FUNCTION_BLOCK WoodBunkEx EXTENDS SectionEx
VAR_IN_OUT
	A21_LSC_C21 : ConveyorLSC;
END_VAR
VAR_IN_OUT
	robotLeft, robotRight : RobotA21;
	toolStorageLeft, toolStorageRight : A21ToolStorage;
	
	stagingTableLeft, stagingTableRight : StagingTable;
	magazineLeft, magazineRight : SkidMagazine;
	
	strapper : StrapMachine;
	
	insertionLeft, insertionRight : Insertion;
	pistonBottom : SimplePiston;
	
	suctionTop : ARRAY[*] OF SuctionPad; (*1..3*)
	suctionLeft : ARRAY[*] OF SuctionPad; (*1..4*)
	suctionRight : ARRAY[*] OF SuctionPad; (*1..4*)
	suctionBottom : ARRAY[*] OF SuctionPad; (*1..2*)
END_VAR
VAR
	conveyorPos : REAL; //may need to move this to SectionEx
	
	step : (IDLE, STAGING, LOAD_WB, PUSH, STRAP, RELEASE, COMPLETE := 1050);
	
	stageStepLeft, stageStepRight : INT;
	loadStepLeft, loadStepRight : INT;
END_VAR
VAR //bundle data
	demoHeight : REAL := 640; //mm
	materialsArr : (*REFERENCE TO*) ARRAY[0..Consts.maxPairs] OF PositionMaterials;
END_VAR
VAR
	//AOIs encapsulate functionality and reduce the number of module variables
	aoiTemplateLeft, aoiTemplateRight : AOI_StagingTemplate;
	aoiStageLeft, aoiStageRight : AOI_StageWoodBunk; 
	aoiLoadLeft, aoiLoadRight : AOI_LoadWoodBunk;
	
	suctionRelease : TON;
	
	//for testing, to be removed when deployoed
	latchLeft, latchRight : BOOL; //prevents SMC sliders from overshooting
	suctionEnableTop, suctionEnableLeft, suctionEnableRight, suctionEnableBottom : BOOL;
END_VAR

aoiBlocks();

SUPER^();

(*
any PackML state-methods that SectionEx has a concrete implementation for will be overriden by concrete FBs that extend it
(ie: all or most of them)

to call the base implementation, add:
	SUPER^.ps_<state>();
to the concrete FB's implementation of that state-method
*)

METHOD PROTECTED aoiBlocks : BOOL
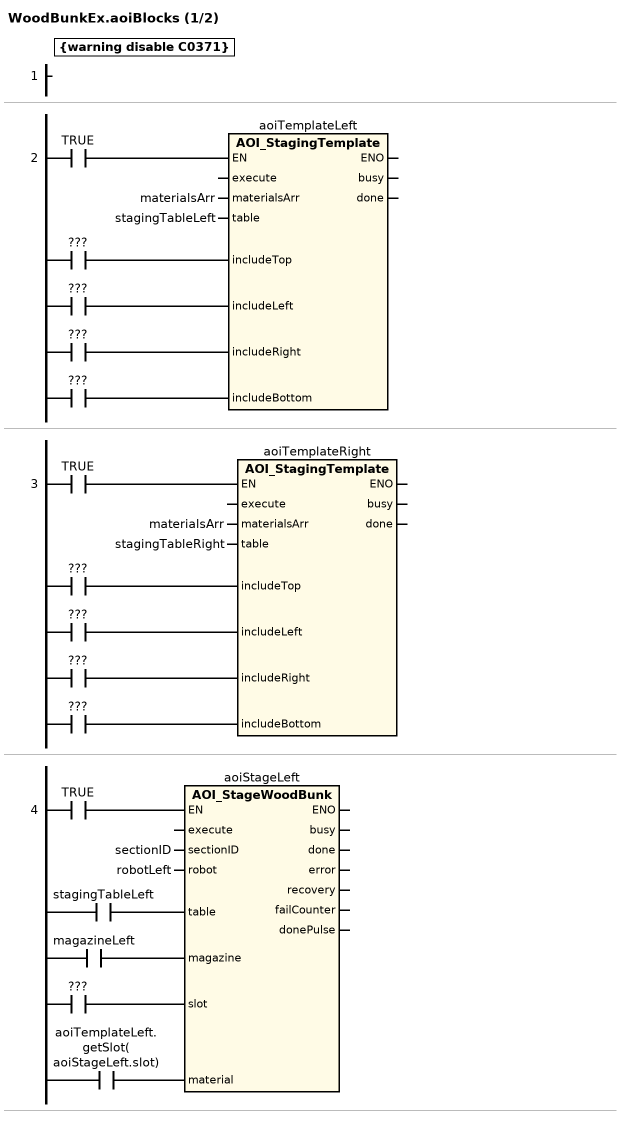
// NETWORK 1
// label: {warning disable C0371}

// NETWORK 2
aoiTemplateLeft(materialsArr := materialsArr, table := stagingTableLeft); // AOI_StagingTemplate

// NETWORK 3
aoiTemplateRight(materialsArr := materialsArr, table := stagingTableRight); // AOI_StagingTemplate

// NETWORK 4
aoiStageLeft(
    sectionID := sectionID,
    robot := robotLeft,
    table := stagingTableLeft,
    magazine := magazineLeft,
    material := aoiTemplateLeft.getSlot(aoiStageLeft.slot)); // AOI_StageWoodBunk

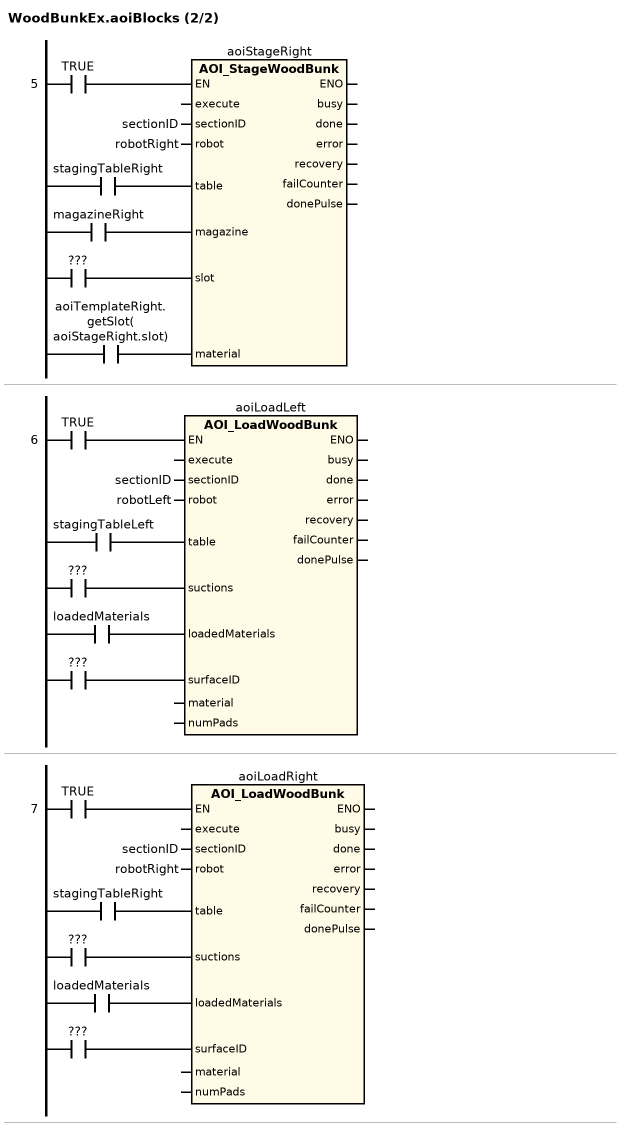
// NETWORK 5
aoiStageRight(
    sectionID := sectionID,
    robot := robotRight,
    table := stagingTableRight,
    magazine := magazineRight,
    material := aoiTemplateRight.getSlot(aoiStageRight.slot)); // AOI_StageWoodBunk

// NETWORK 6
aoiLoadLeft(
    sectionID := sectionID,
    robot := robotLeft,
    table := stagingTableLeft,
    loadedMaterials := loadedMaterials); // AOI_LoadWoodBunk

// NETWORK 7
aoiLoadRight(
    sectionID := sectionID,
    robot := robotRight,
    table := stagingTableRight,
    loadedMaterials := loadedMaterials); // AOI_LoadWoodBunk
END_METHOD

METHOD PROTECTED load : BOOL
VAR_INPUT
	pairIndex : INT;
END_VAR
VAR_OUTPUT
	error : BOOL;
END_VAR
VAR
	pair : REFERENCE TO PositionMaterials REF= materialsArr[pairIndex];
	errorLeft, errorRight : BOOL;
END_VAR
{warning disable C0371}
(*
this is the new code for loading wood bunks from staging table to insertion
loading sequences are independent as each side has its own step variable
can be extended by changing the include<> parameters
*)

load :=
	loadEx(
		robot:= robotLeft, 
		aoiLoad:= aoiLoadLeft, 
		loadStep:= loadStepLeft, 
		pairIndex:= pairIndex, 
		includeTop:= TRUE, 
		includeLeft:= TRUE, 
		includeRight:= FALSE, 
		includeBottom:= FALSE, 
		error=> errorLeft)
	AND
	loadEx(
		robot:= robotRight, 
		aoiLoad:= aoiLoadRight, 
		loadStep:= loadStepRight, 
		pairIndex:= pairIndex, 
		includeTop:= FALSE, 
		includeLeft:= FALSE, 
		includeRight:= TRUE, 
		includeBottom:= TRUE, 
		error=> errorRight);
		
error := errorLeft OR errorRight;

(*
below is the old code for loading wood bunks from staging table to insertion
it loads wood bunks in sets - top/bottom, then sides
if one side is finished loading a set before the other, it waits until the other side is done before advancing the set
*)
(*
IF robotLeft.error OR robotRight.error THEN
	error := TRUE;
	RETURN;
	
ELSIF 
	(robotLeft.reservation <> sectionID AND_THEN NOT robotLeft.reserve(sectionID)) OR 
	(robotRight.reservation <> sectionID AND_THEN NOT robotRight.reserve(sectionID))
THEN //loading requires both robots be reserved together
	RETURN;
	
ELSIF //robots have wrong tool
	(robotLeft.tool <> sectionID AND_THEN NOT robotLeft.changeEOAT(targetTool := sectionID)) OR
	(robotRight.tool <> sectionID AND_THEN NOT robotRight.changeEOAT(targetTool := sectionID))
THEN
	RETURN;
	
END_IF

CASE loadStep OF
	0: //top and bottom
		IF aoiLoadLeft.done AND aoiLoadRight.done THEN
			aoiLoadLeft.execute := aoiLoadRight.execute := FALSE;
			aoiLoadLeft.material := aoiLoadRight.material := '';
			
			aoiLoadLeft.reset();
			aoiLoadRight.reset();
			loadStep := 10;
			RETURN;
		END_IF
		
		aoiLoadLeft.suctions := suctionTop;
		aoiLoadLeft.surfaceID := Surface.TOP;
		aoiLoadLeft.material := pair.top;
		aoiLoadLeft.numPads := UPPER_BOUND(suctionTop, 1) - LOWER_BOUND(suctionTop, 1) + 1;
		
		aoiLoadRight.suctions := suctionBottom;
		aoiLoadRight.surfaceID := Surface.BOTTOM;
		aoiLoadRight.material := pair.bottom;
		aoiLoadRight.numPads := UPPER_BOUND(suctionBottom, 1) - LOWER_BOUND(suctionBottom, 1) + 1;
		
		aoiLoadLeft.execute := NOT aoiLoadLeft.done AND NOT aoiLoadLeft.busy;
		aoiLoadRight.execute := NOT aoiLoadRight.done AND NOT aoiLoadRight.busy;
		
	10: //sides
		IF aoiLoadLeft.done AND aoiLoadRight.done THEN
			aoiLoadLeft.execute := aoiLoadRight.execute := FALSE;
			aoiLoadLeft.material := aoiLoadRight.material := '';
			
			aoiLoadLeft.reset();
			aoiLoadRight.reset();
			loadStep := COMPLETE;
			RETURN;
		END_IF
		
		aoiLoadLeft.suctions := suctionLeft;
		aoiLoadLeft.surfaceID := Surface.LEFT;
		aoiLoadLeft.material := pair.left;
		aoiLoadLeft.numPads := UPPER_BOUND(suctionLeft, 1) - LOWER_BOUND(suctionLeft, 1) + 1;
		
		aoiLoadRight.suctions := suctionRight;
		aoiLoadRight.surfaceID := Surface.RIGHT;
		aoiLoadRight.material := pair.right;
		aoiLoadRight.numPads := UPPER_BOUND(suctionRight, 1) - LOWER_BOUND(suctionRight, 1) + 1;
		
		aoiLoadLeft.execute := NOT aoiLoadLeft.done AND NOT aoiLoadLeft.busy;
		aoiLoadRight.execute := NOT aoiLoadRight.done AND NOT aoiLoadRight.busy;
		
	COMPLETE:				
		robotLeft.release(sectionID);
		robotRight.release(sectionID);
		
		aoiLoadLeft.material := aoiLoadRight.material := '';
		aoiLoadLeft.execute := aoiLoadRight.execute := FALSE;
		
		loadStep := 0;
		load := TRUE;
END_CASE

//--------------------------------------------------
IF aoiLoadLeft.recovery THEN //if loading in recovery mode - refill table, resume loading when finished
	aoiLoadLeft.execute := stageEx(
		robot:= robotLeft, 
		aoiTemplate:= aoiTemplateLeft, 
		aoiStaging:= aoiStageLeft, 
		stageStep:= stageStepLeft, 
		includeTop:= TRUE, 
		includeLeft:= TRUE, 
		includeRight:= FALSE, 
		includeBottom:= FALSE, 
		error=> );
ELSE
	//loadLeft.execute := NOT loadLeft.busy AND NOT loadLeft.done;
END_IF
//--------------------------------------------------
IF aoiLoadRight.recovery THEN
	aoiLoadRight.execute := stageEx(
		robot:= robotRight, 
		aoiTemplate:= aoiTemplateRight, 
		aoiStaging:= aoiStageRight, 
		stageStep:= stageStepRight, 
		includeTop:= FALSE, 
		includeLeft:= FALSE, 
		includeRight:= TRUE, 
		includeBottom:= TRUE, 
		error=> );
ELSE
	//loadRight.execute := NOT loadRight.busy AND NOT loadRight.done;
END_IF
//--------------------------------------------------
	
error := aoiLoadLeft.error OR aoiLoadRight.error;
*)
END_METHOD

METHOD PRIVATE loadEx : BOOL
VAR_IN_OUT
	robot : RobotA21;
	aoiLoad : AOI_LoadWoodBunk;
	loadStep : INT;
END_VAR
VAR_INPUT
	pairIndex : INT;
	includeTop, includeLeft, includeRight, includeBottom : BOOL;
END_VAR
VAR_OUTPUT
	error : BOOL;
END_VAR
VAR
	pair : REFERENCE TO PositionMaterials REF= materialsArr[pairIndex];
END_VAR
{warning disable C0371}
IF robot.error THEN
	error := TRUE;
	RETURN;
ELSIF robot.reservation <> sectionID AND_THEN NOT robot.reserve(sectionID) THEN
	RETURN;
ELSIF robot.tool <> sectionID AND_THEN NOT robot.changeEOAT(targetTool := sectionID) THEN
	RETURN;
END_IF

error := aoiLoad.error;

CASE loadStep OF
	0:
		loadStep := Surface.TOP;
	
	Surface.TOP:		
		IF NOT includeTop OR aoiLoad.donePulse THEN
			aoiLoad.execute := FALSE;
			aoiLoad.material := '';
			loadStep := Surface.BOTTOM;
			RETURN;
		END_IF
		
		aoiLoad.surfaceID := Surface.TOP;
		aoiLoad.material := pair.top;
		aoiLoad.suctions := suctionTop;
		aoiLoad.numPads := UPPER_BOUND(suctionTop, 1) - LOWER_BOUND(suctionTop, 1) + 1;
		
		aoiLoad.execute := NOT aoiLoad.busy;
		
	Surface.BOTTOM:
		IF NOT includeBottom OR aoiLoad.donePulse THEN
			aoiLoad.execute := FALSE;
			aoiLoad.material := '';
			loadStep := Surface.LEFT;
			RETURN;
		END_IF
		
		aoiLoad.surfaceID := Surface.BOTTOM;
		aoiLoad.material := pair.bottom;
		aoiLoad.suctions := suctionBottom;
		aoiLoad.numPads := UPPER_BOUND(suctionBottom, 1) - LOWER_BOUND(suctionBottom, 1) + 1;
		
		aoiLoad.execute := NOT aoiLoad.busy;
		
	Surface.LEFT:
		IF NOT includeLeft OR aoiLoad.donePulse THEN
			aoiLoad.execute := FALSE;
			aoiLoad.material := '';
			loadStep := Surface.RIGHT;
			RETURN;
		END_IF
		
		aoiLoad.surfaceID := Surface.LEFT;
		aoiLoad.material := pair.left;
		aoiLoad.suctions := suctionLeft;
		aoiLoad.numPads := UPPER_BOUND(suctionLeft, 1) - LOWER_BOUND(suctionLeft, 1) + 1;
		
		aoiLoad.execute := NOT aoiLoad.busy;
		
	Surface.RIGHT:
		IF NOT includeRight OR aoiLoad.donePulse THEN
			aoiLoad.execute := FALSE;
			aoiLoad.material := '';
			loadStep := COMPLETE;
			RETURN;
		END_IF
		
		aoiLoad.surfaceID := Surface.RIGHT;
		aoiLoad.material := pair.right;
		aoiLoad.suctions := suctionRight;
		aoiLoad.numPads := UPPER_BOUND(suctionRight, 1) - LOWER_BOUND(suctionRight, 1) + 1;
		
		aoiLoad.execute := NOT aoiLoad.busy;
		
	COMPLETE:				
		robot.release(sectionID);
		
		aoiLoad.material := '';
		aoiLoad.execute := FALSE;
		
		loadEx := TRUE;
END_CASE
END_METHOD

METHOD PROTECTED maintenance : BOOL
VAR_INPUT
END_VAR
{warning disable C0371}
//no specific tasks yet, free run and testing
SetSuctions(suctionTop, suctionEnableTop);
SetSuctions(suctionLeft, suctionEnableLeft);
SetSuctions(suctionRight, suctionEnableRight);
SetSuctions(suctionBottom, suctionEnableBottom);

IF robotLeft.Done THEN
	robotLeft.clearCommand();
END_IF

IF robotRight.Done THEN
	robotRight.clearCommand();
END_IF
END_METHOD

METHOD PROTECTED manual : BOOL
VAR_INPUT
END_VAR
END_METHOD

METHOD PROTECTED process : BOOL
VAR_INPUT
	auto : BOOL;
END_VAR
VAR_OUTPUT
	error : BOOL;
END_VAR
VAR
	currentPair : REFERENCE TO PositionMaterials REF= materialsArr[iPair];
END_VAR
{warning disable C0371}
IF iPair >= Consts.maxPairs THEN
	process := TRUE;
	RETURN;
ELSIF NOT PositionIsValid(pair := currentPair) THEN
	iPair := iPair + 1;
	RETURN;
END_IF

CASE step OF
	IDLE:
		IF auto OR_ELSE execute THEN
			step := STAGING;
		END_IF

	LOAD_WB:
		IF
			directionCheckAndSet(conveyorPos, currentPair.position) AND 
			( (auto AND done) OR_ELSE (NOT auto AND execute) )
		THEN
			robotLeft.clearCommand();
			robotRight.clearCommand();
			
			aoiLoadLeft.reset();
			aoiLoadRight.reset();
			
			loadStepLeft := loadStepRight := 0;
			stageStepLeft := stageStepRight := 0;
			
			done := FALSE;
			suctionEnableTop := suctionEnableLeft := suctionEnableRight := suctionEnableBottom := FALSE;
			execute := FALSE;
			
			step := PUSH;
			RETURN;
		END_IF
		
		IF NOT done THEN
			done := load(pairIndex := iPair, error => error);
		END_IF
		
		IF NOT auto THEN
			SetSuctions(suctionTop, suctionEnableTop);
			SetSuctions(suctionLeft, suctionEnableLeft);
			SetSuctions(suctionRight, suctionEnableRight);
			SetSuctions(suctionBottom, suctionEnableBottom);
		END_IF
		
	PUSH:
		IF
			(auto AND latchLeft AND latchRight AND pistonBottom.extended) OR_ELSE
			(NOT auto AND execute)
		THEN
			insertionLeft.stop();
			insertionRight.stop();
			
			latchLeft := latchRight := FALSE;
			execute := FALSE;
			step := STRAP;
			RETURN;
		END_IF
		
		IF NOT validateInsertion(checkTop:= FALSE, checkLeft:= FALSE, checkRight:= FALSE, checkBottom:= FALSE) THEN
			error := TRUE;
			RETURN;
		END_IF
		
		IF 
			insertionLeft.sliderPos <> demoHeight/2 OR 
			insertionRight.sliderPos <> demoHeight/2
		THEN
			insertionLeft.align(demoHeight/2);
			insertionRight.align(demoHeight/2);
			RETURN;
		END_IF
		
		
		IF insertionLeft.Contact THEN
			latchLeft := TRUE;
		ELSIF NOT latchLeft THEN
			insertionLeft.press();
		END_IF
		
		IF insertionRight.Contact THEN
			latchRight := TRUE;
		ELSIF NOT latchRight THEN
			insertionRight.press();
		END_IF
		pistonBottom.extend();
		
	STRAP:
		suctionRelease(IN:= , PT:= suctionReleaseDelay, Q=> , ET=> );
		
		strapper.bEnable := TRUE;
		IF strapper.done THEN
			suctionRelease.IN := FALSE;
			step := RELEASE;
			RETURN;
		END_IF
		
		IF suctionRelease.Q THEN
			SetSuctions(suctionTop, FALSE);
			SetSuctions(suctionLeft, FALSE);
			SetSuctions(suctionRight, FALSE);
			SetSuctions(suctionBottom, FALSE);
		ELSIF strapper.atBundleLevel THEN
			suctionRelease.IN := TRUE;
		END_IF
		
		IF strapper.ready THEN
			strapper.strap();
		END_IF
		
		IF execute THEN
			suctionRelease.IN := FALSE;
			execute := FALSE;
			step := RELEASE;
		END_IF
		
	RELEASE: //release command		
		insertionLeft.toHome();
		insertionRight.toHome();
		pistonBottom.retract();
		
		IF 
			(insertionLeft.screw.AtHome AND insertionRight.screw.AtHome AND pistonBottom.retracted) OR
			execute
		THEN
			execute := FALSE;
			step := COMPLETE;
		END_IF
	
	COMPLETE:
		//reset everything
		iPair := iPair + 1;
		step := IDLE;
END_CASE
END_METHOD

METHOD PROTECTED ps_AbortCondition : BOOL
VAR_INPUT
END_VAR
{warning disable C0371}
ps_AbortCondition :=
	insertionLeft.error OR 
	insertionRight.error OR 
	robotLeft.error OR 
	robotRight.error OR
	strapper.error;
END_METHOD

METHOD PROTECTED ps_Aborted : BOOL
VAR_INPUT
END_VAR
ps_Aborted := TRUE;
END_METHOD

METHOD PROTECTED ps_Aborting : BOOL
VAR_INPUT
END_VAR
{warning disable C0371}
insertionLeft.stop();
insertionRight.stop();
pistonBottom.stop();

aoiLoadLeft.reset();
aoiLoadRight.reset();

aoiStageLeft.reset();
aoiStageRight.reset();

robotLeft.clearCommand();
robotRight.clearCommand();

//stop conveyors

ps_Aborting :=
	NOT insertionLeft.active AND
	NOT insertionRight.active AND
	NOT pistonBottom.busy AND
	NOT robotLeft.Busy AND
	NOT robotRight.Busy;
END_METHOD

METHOD PROTECTED ps_Clearing : BOOL
VAR_INPUT
END_VAR
{warning disable C0371}
insertionLeft.reset();
insertionRight.reset();

ps_Clearing := 
	NOT insertionLeft.error AND
	NOT insertionRight.error AND
	NOT strapper.error AND
	NOT robotLeft.error AND
	NOT robotRight.error;
END_METHOD

METHOD PROTECTED ps_Complete : BOOL
VAR_INPUT
END_VAR
ps_Complete := TRUE;
END_METHOD

METHOD PROTECTED ps_Completing : BOOL
VAR_INPUT
END_VAR
ps_Completing := NOT occupied;
END_METHOD

METHOD PROTECTED ps_Execute : BOOL
VAR_INPUT
END_VAR
VAR_OUTPUT
	error : BOOL;
END_VAR
SUPER^.ps_Execute();
END_METHOD

METHOD PROTECTED ps_Held : BOOL
VAR_INPUT
END_VAR
ps_Held := NOT hold;
END_METHOD

METHOD PROTECTED ps_HoldCondition : BOOL
VAR_INPUT
END_VAR
END_METHOD

METHOD PROTECTED ps_Holding : BOOL
VAR_INPUT
END_VAR
{warning disable C0371}
insertionLeft.stop();
insertionRight.stop();
pistonBottom.stop();
//set robot to pause

ps_Holding :=
	NOT insertionLeft.active AND
	NOT insertionRight.active;
END_METHOD

METHOD PROTECTED ps_Idle : BOOL
VAR_INPUT
END_VAR
ps_Idle := execute;
execute := FALSE;
END_METHOD

METHOD PROTECTED ps_Resetting : BOOL
VAR_INPUT
END_VAR
{warning disable C0371}
insertionLeft.reset();
insertionRight.reset();

ps_Resetting := 
	reset AND
	NOT insertionLeft.error AND
	NOT insertionRight.error AND
	NOT strapper.error AND
	NOT robotLeft.error AND
	NOT robotRight.error;
END_METHOD

METHOD PROTECTED ps_Starting : BOOL
VAR_INPUT
END_VAR
{warning disable C0371}
robotLeft.clearCommand();
robotRight.clearCommand();

insertionLeft.homingSequence();
insertionRight.homingSequence();
pistonBottom.retract();

ps_Starting := 
	insertionLeft.screw.HomeSet AND 
	insertionRight.screw.HomeSet AND 
	pistonBottom.retracted;
END_METHOD

METHOD PROTECTED ps_StopCondition : BOOL
VAR_INPUT
END_VAR
ps_StopCondition := 
	stop;
END_METHOD

METHOD PROTECTED ps_Stopped : BOOL
VAR_INPUT
END_VAR
ps_Stopped := TRUE;
END_METHOD

METHOD PROTECTED ps_Stopping : BOOL
VAR_INPUT
END_VAR
{warning disable C0371}
insertionLeft.stop();
insertionRight.stop();
pistonBottom.stop();

aoiLoadLeft.reset();
aoiLoadRight.reset();

aoiStageLeft.reset();
aoiStageRight.reset();

robotLeft.clearCommand();
robotRight.clearCommand();

//stop conveyors

ps_Stopping :=
	NOT insertionLeft.active AND
	NOT insertionRight.active AND
	NOT pistonBottom.busy AND
	NOT robotLeft.Busy AND
	NOT robotRight.Busy;
END_METHOD

METHOD PROTECTED ps_SuspendCondition : BOOL
VAR_INPUT
END_VAR
END_METHOD

METHOD PROTECTED ps_Suspended : BOOL
VAR_INPUT
END_VAR
ps_Suspended := NOT ps_SuspendCondition();
END_METHOD

METHOD PROTECTED ps_Suspending : BOOL
VAR_INPUT
END_VAR
ps_Suspending := TRUE;
END_METHOD

METHOD PROTECTED ps_Unholding : BOOL
VAR_INPUT
END_VAR
ps_Unholding := TRUE;
END_METHOD

METHOD PROTECTED ps_Unsuspending : BOOL
VAR_INPUT
END_VAR
ps_Unsuspending := TRUE;
END_METHOD

METHOD PROTECTED FINAL runSectionTasks : BOOL
VAR_INPUT
	auto : BOOL;
END_VAR
VAR_OUTPUT
	error : BOOL;
END_VAR
SUPER^.runSectionTasks(auto := auto, error => error);

CASE status OF //add additional instructions for each state
	SectionTask.IDLE:
		//
	
	SectionTask.ALIGNING:
		stage(error => error);
		
	SectionTask.ACTIVE:
		//
		
	SectionTask.CLEARING:
		aoiLoadLeft.reset();
		aoiLoadRight.reset();
		
		aoiStageLeft.reset();
		aoiStageRight.reset();
		
		aoiTemplateLeft.reset();
		aoiTemplateRight.reset();
		
	SectionTask.COMPLETE:	
		//
		
	-100:
		//
		
END_CASE
END_METHOD

METHOD PROTECTED stage : BOOL
VAR_OUTPUT
	error : BOOL;
END_VAR
{warning disable C0371}

(*
this method only exists to call stageEx() for both robots
*)
(*
stage := leftDone AND rightDone;

IF NOT leftDone THEN
	leftDone := stageEx(
		robot:= robotLeft, 
		aoiTemplate:= aoiTemplateLeft, 
		aoiStaging:= aoiStageLeft, 
		stageStep:= stageStepLeft, 
		//iSlot:= iSlotLeft, 
		includeTop:= TRUE, 
		includeLeft:= TRUE, 
		includeRight:= FALSE, 
		includeBottom:= FALSE, 
		error=> );
END_IF

IF NOT rightDone THEN
	rightDone := stageEx(
		robot:= robotRight, 
		aoiTemplate:= aoiTemplateRight, 
		aoiStaging:= aoiStageRight, 
		stageStep:= stageStepRight, 
		//iSlot:= iSlotRight, 
		includeTop:= FALSE, 
		includeLeft:= FALSE, 
		includeRight:= TRUE, 
		includeBottom:= TRUE, 
		error=> );
END_IF
*)

stage := 
	stageEx(
		robot:= robotLeft, 
		aoiTemplate:= aoiTemplateLeft, 
		aoiStaging:= aoiStageLeft, 
		stageStep:= stageStepLeft, 
		includeTop:= TRUE, 
		includeLeft:= TRUE, 
		includeRight:= FALSE, 
		includeBottom:= FALSE, 
		error=> )
	AND
	stageEx(
		robot:= robotRight, 
		aoiTemplate:= aoiTemplateRight, 
		aoiStaging:= aoiStageRight, 
		stageStep:= stageStepRight, 
		includeTop:= FALSE, 
		includeLeft:= FALSE, 
		includeRight:= TRUE, 
		includeBottom:= TRUE, 
		error=> );
END_METHOD

METHOD PRIVATE stageEx : BOOL
VAR_IN_OUT
	robot : RobotA21;
	aoiTemplate : AOI_StagingTemplate;
	aoiStaging : AOI_StageWoodBunk;
	stageStep : INT;
END_VAR
VAR_INPUT
	includeTop, includeLeft, includeRight, includeBottom : BOOL;
END_VAR
VAR_OUTPUT
	error : BOOL;
END_VAR
{warning disable C0371}
IF robot.error THEN
	error := TRUE;
	RETURN;
ELSIF robot.reservation <> sectionID AND_THEN NOT robot.reserve(sectionID) THEN
	RETURN;
ELSIF robot.tool <> sectionID AND_THEN NOT robot.changeEOAT(targetTool := sectionID) THEN
	RETURN;
END_IF

CASE stageStep OF
	0: //generate staging template
		IF aoiTemplate.done THEN
			aoiTemplate.execute := FALSE;
			stageStep := 10;
			RETURN;
		END_IF
		
		aoiTemplate.execute := NOT aoiTemplate.busy;
		
		aoiTemplate.includeTop := includeTop;
		aoiTemplate.includeLeft := includeLeft;
		aoiTemplate.includeRight := includeRight;
		aoiTemplate.includeBottom := includeBottom;
		
	10: //stage tables
		IF aoiStaging.slot > 10 THEN
			aoiStaging.execute := FALSE;			
			stageStep := COMPLETE;
			RETURN;
		END_IF
		
		aoiStaging.execute := NOT aoiStaging.busy; //execute if aoiStaging is ready
		
		aoiStaging.slot := MAX(1, aoiStaging.slot); //if 0, sets to 1
		aoiStaging.slot := MIN(aoiStaging.slot, 999); //prevents overflow 
		
		IF aoiStaging.donePulse THEN
			aoiStaging.slot := aoiStaging.slot + 1;
		END_IF
	
	COMPLETE:
		aoiTemplate.clearTemplate();
		aoiTemplate.execute := FALSE;
		aoiStaging.execute := FALSE;
		aoiStaging.reset();
		
		robot.release(sectionID);
		
		aoiStaging.slot := 0;
		
		stageEx := TRUE;
		//stageStep := 0;
END_CASE

error := aoiStaging.error;
END_METHOD

METHOD PROTECTED unload : BOOL
VAR_INPUT
END_VAR
//unload from insertion
//remove from staging table
END_METHOD

METHOD PROTECTED validateInsertion : BOOL
VAR_INPUT
	checkTop : BOOL;
	checkLeft : BOOL;
	checkRight : BOOL;
	checkBottom : BOOL;
END_VAR
validateInsertion := 
	(NOT checkTop OR_ELSE SuctionQuality(suctions:= suctionTop)) AND
	(NOT checkLeft OR_ELSE SuctionQuality(suctions:= suctionLeft)) AND
	(NOT checkRight OR_ELSE SuctionQuality(suctions:= suctionRight)) AND
	(NOT checkBottom OR_ELSE SuctionQuality(suctions:= suctionBottom));

(*
validateSuctionQuality := 
	(
		NOT checkTop OR_ELSE InsertionQuality(
			suctions:= suctionTop, 
			insertionMaterial:= loadedMaterials[Surface.TOP], 
			recipeMaterial:= materialsArr[iPair].top)
	) AND
	(
		NOT checkLeft OR_ELSE InsertionQuality(
			suctions:= suctionLeft, 
			insertionMaterial:= loadedMaterials[Surface.LEFT], 
			recipeMaterial:= materialsArr[iPair].left)
	) AND
	(
		NOT checkRight OR_ELSE InsertionQuality(
			suctions:= suctionRight, 
			insertionMaterial:= loadedMaterials[Surface.RIGHT], 
			recipeMaterial:= materialsArr[iPair].right)
	) AND
	(
		NOT checkBottom OR_ELSE InsertionQuality(
			suctions:= suctionBottom, 
			insertionMaterial:= loadedMaterials[Surface.BOTTOM], 
			recipeMaterial:= materialsArr[iPair].bottom)
	);
*)
END_METHOD

END_FUNCTION_BLOCK

(* stored: Version 1.1.0.1, ProductVersion 3.1.4024.11
   POU WoodBunkEx: Id {7c192e4b-e9ee-4c1c-a070-15e2c6191789}, SpecialFunc None
   Folder Actions_Cyclic: Id {4a4594ef-dea4-4aa0-b286-04c344ad8bce}
   Folder PML Conditions: Id {c72861c0-c0ce-4674-aeb2-9bafbcf1ffb2}
   Folder PML States: Id {bb7e80d1-aaba-45a3-942d-4c0ae1b7e0a1}
   Folder TaskEx: Id {5b3fc18f-f550-457a-8a17-1d786d7a73b0}
   Method aoiBlocks: Id {8c2b7778-065d-411a-81bc-dde8062443b8}
   Method load: Id {41d6aef3-60c1-439a-bdd2-e372cfed0011}
   Method loadEx: Id {26e40d6d-60a4-4c2c-bba4-a7493624a410}
   Method maintenance: Id {3ded9c42-31de-4c46-b6b2-588795d0455a}
   Method manual: Id {0c3f7a60-10c4-482a-82e7-c6357c99d1f0}
   Method process: Id {125184ca-77bd-471a-a90f-30ac270f7324}
   Method ps_AbortCondition: Id {79544249-b19f-4b65-805e-588b9e65f109}
   Method ps_Aborted: Id {b0b87d9a-5af9-4b16-b799-62759d97cc29}
   Method ps_Aborting: Id {d369707c-28f8-4c64-966f-5bb6a3587ba5}
   Method ps_Clearing: Id {b1bcfdaf-5358-4ace-937d-293bb0c837c2}
   Method ps_Complete: Id {164491d5-8f7b-4481-a463-d014092e154c}
   Method ps_Completing: Id {890e9e7f-1dec-47cc-9e28-3b0a8d0719a2}
   Method ps_Execute: Id {53c1cce1-52a2-4557-8c8e-c609d5374b63}
   Method ps_Held: Id {9d7440d6-bc19-48cc-b67b-cef2292c495c}
   Method ps_HoldCondition: Id {7e586a9c-7b49-4afa-b286-4520d00847aa}
   Method ps_Holding: Id {9c0c96db-5709-4873-af32-26d4591962e1}
   Method ps_Idle: Id {628c7b09-fba5-4346-a13d-9dfc0dc54180}
   Method ps_Resetting: Id {ed7fb93f-1f68-484d-bf76-f2c9f1db3c72}
   Method ps_Starting: Id {7764a973-763c-4f51-8655-e151dbd80f89}
   Method ps_StopCondition: Id {b05bc17a-c428-4e6e-8ce7-2886a0e44766}
   Method ps_Stopped: Id {77d4cc84-065a-404e-b8b7-156c1902e0aa}
   Method ps_Stopping: Id {194f87af-0f78-4bc2-825a-74091d7c1f8d}
   Method ps_SuspendCondition: Id {17d92194-540a-41ca-bb52-08b0d05a6c82}
   Method ps_Suspended: Id {377e7b77-6b80-441b-9846-1f4cf89cd039}
   Method ps_Suspending: Id {7c542666-c215-405f-bec8-290880091086}
   Method ps_Unholding: Id {f2bcee8f-48f1-4152-804e-2779a6c303f5}
   Method ps_Unsuspending: Id {a0abdd12-97e3-4749-8a59-2082fe193f70}
   Method runSectionTasks: Id {b1351305-e851-4156-92d6-e8291baa67e7}
   Method stage: Id {394ea3b0-a477-4afc-b551-89e83b2984a7}
   Method stageEx: Id {5592989f-862c-4d1d-a10b-2f36f2ccb694}
   Method unload: Id {1238b592-1050-41d7-99da-ccbfe9e4fae5}
   Method validateInsertion: Id {b1904323-60a7-4bcf-ac74-c2042e21b0b7} *)
